RoboDK station: ALTERNATIVA 2 - PYTHON.rdk

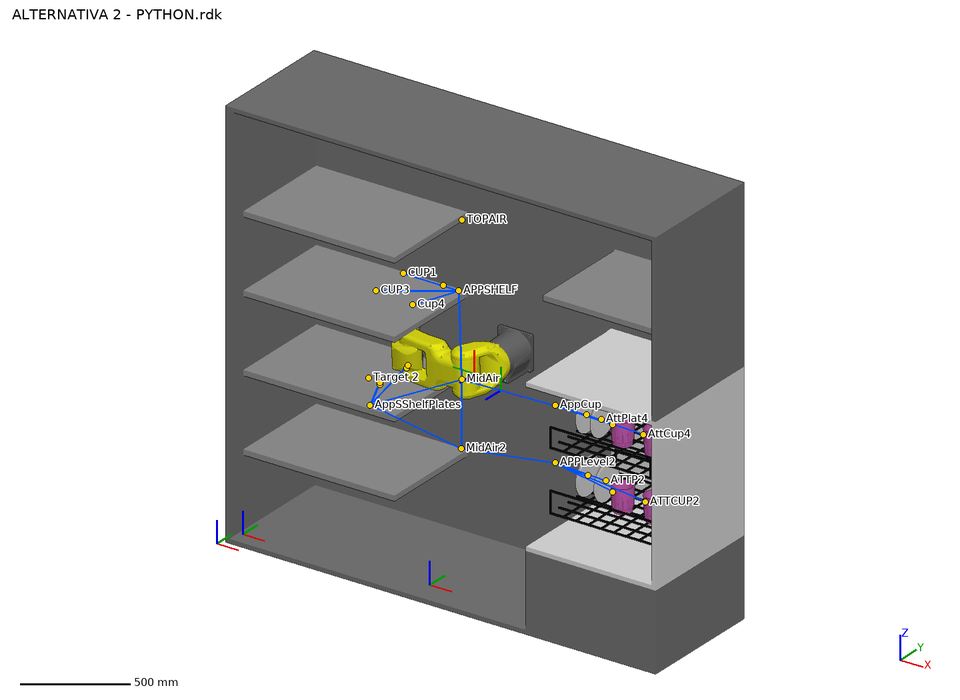
[picture v0: the station drawn from its stored meshes, robots at their saved joint values, targets as dots, program paths as lines]
Station ALTERNATIVA 2 (saved by RoboDK 6.0.0). Poses are relative to the parent item; angles as X-Y-Z fixed-axis rotations.
  - object modelo_solo_interior_v6 at (0, 0, 0) mm, size 2380 x 700 x 2200 mm, geometry from modelo_solo_interior_v6.obj
  - frame MUEBLE  at (-14.91, -46.19, 5.82) mm
  - frame Fanuc LR Mate 200iD Base at (1300, 320, 1000) mm, rotated rx 90 ry 0 rz 0 deg
    - object VASO_2 at (880, -75, 20) mm, size 110.6 x 132.4 x 110.6 mm, geometry from glass-obj.obj
  - frame Frame 3 at (80, 23.81, 50) mm
    - frame My Mechanism Base at (1040, -6.19, 40) mm
      - robot My Mechanism: 1 axes
          modified DH rows (alpha deg, a mm, theta deg, d mm): 0, 0, 0, 0 linear
          base shift (0, 0, 0) mm, rotated rx 180 ry 0 rz 180 deg
          joint limits [0] to [1500]; home [0]; saved at [905.84]
        - frame Fanuc LR Mate 200iD Base at (-120, 180, 120) mm, rotated rx -90 ry 0 rz -180 deg
          - robot Fanuc LR Mate 200iD: 6 axes, payload 7 kg, reach 717 mm, repeatability 0.02 mm, weight 25 kg
              modified DH rows (alpha deg, a mm, theta deg, d mm): 0, 0, 0, 330; -90, 50, -90, 0; 0, 330, 0, 0; -90, 35, 0, 335; 90, 0, 0, 0; -90, 0, 0, 80
              base shift (0, 0, -330) mm
              joint limits [-170, -100, -67, -190, -125, -360] to [170, 145, 213, 190, 124, 360]; home [0, 0, 0, 0, 0, 0]; saved at [93.044, 96.293, -58.546, 87.403, 88.412, -211.418]
            - tool RobotiQ EPick Vacuum Gripper (1 Cup), TCP at (0, 0, 130) mm, size 75 x 83 x 136.1 mm
    - target AttCup4 (Cartesian target) at (2025.95, 272.71, 963.12) mm, rotated rx 90.33 ry 1.97 rz 94.86 deg; joints [-104.637, 115.612, 4.554, 123.155, 17.105, 58.882, 975.84] of Fanuc LR Mate 200iD
    - target AppCup (Cartesian target) at (1576.89, 214.64, 1005.7) mm, rotated rx 96.54 ry 1.97 rz 94.86 deg; joints [-118.032, 21.715, -84.906, 21.706, 80.662, 180.626, 980.84] of Fanuc LR Mate 200iD
    - target Target 2 (Cartesian target) at (718.15, -32.51, 1004.9) mm, rotated rx -83.96 ry 1.97 rz 94.86 deg; joints [109.561, -20.769, -26.684, -42.184, 39.93, -145.464, 905.84] of Fanuc LR Mate 200iD
    - target MidAir (Cartesian target) at (1233.73, -32.54, 1140.54) mm, rotated rx 23.3 ry -5.22 rz 90.43 deg; joints [2.19, -20.76, -26.68, -42.18, 39.92, -145.46, 540.58] of Fanuc LR Mate 200iD
    - target ATTCup3 (Cartesian target) at (1855.95, 272.71, 963.12) mm, rotated rx 90.33 ry 1.97 rz 94.86 deg; joints [-109.413, 54.482, -60.076, 22.825, 57.115, 170.802, 975.84] of Fanuc LR Mate 200iD
    - target AttPlat4 (Cartesian target) at (1791.95, 272.71, 973.12) mm, rotated rx 90.33 ry 1.97 rz 94.86 deg; joints [-110.912, 48.655, -68.61, 22.691, 65.237, 173.884, 975.84] of Fanuc LR Mate 200iD
    - target AttP3 (Cartesian target) at (1710.95, 272.71, 973.12) mm, rotated rx 90.33 ry 1.97 rz 94.86 deg; joints [-115.299, 43.34, -78.431, 25.854, 74.698, 176.966, 975.84] of Fanuc LR Mate 200iD
    - target ATTCUP2 (Cartesian target) at (2035.98, 272.65, 625.36) mm, rotated rx 90.33 ry 1.97 rz 94.86 deg; joints [-104.42, 81.896, -28.227, 32.378, 26.939, 153.732, 637.99] of Fanuc LR Mate 200iD
    - target ATTCUP1 (Cartesian target) at (1855.94, 272.75, 625.32) mm, rotated rx 90.32 ry 1.97 rz 94.87 deg; joints [-109.41, 54.48, -60.08, 22.831, 57.11, 170.799, 637.99] of Fanuc LR Mate 200iD
    - target ATTP2 (Cartesian target) at (1811.98, 282.72, 665.28) mm, rotated rx 90.33 ry 1.97 rz 94.85 deg; joints [-106.543, 51.004, -68.493, 17.943, 64.576, 175.489, 637.99] of Fanuc LR Mate 200iD
    - target ATTP1 (Cartesian target) at (1711.98, 282.72, 665.28) mm, rotated rx 90.33 ry 1.97 rz 94.85 deg; joints [-110.992, 44.665, -81.327, 21.149, 77.053, 178.867, 637.99] of Fanuc LR Mate 200iD
    - target APPLevel2 (Cartesian target) at (1576.9, 214.61, 716.41) mm, rotated rx 96.54 ry 1.97 rz 94.85 deg; joints [-118.03, 21.71, -84.9, 21.7, 80.66, 180.62, 691.56] of Fanuc LR Mate 200iD
    - target CUP1 (Cartesian target) at (548.14, 487.49, 1274.9) mm, rotated rx 90 ry 0 rz -90 deg; joints [120.418, 87.929, -81.134, -30.72, 82.362, 4.516, 1350.84] of Fanuc LR Mate 200iD
    - target MidAir2 (Cartesian target) at (1233.71, -32.66, 789.98) mm, rotated rx 23.3 ry -5.22 rz 90.42 deg; joints [2.19, -20.75, -26.67, -42.17, 39.92, -145.45, 189.94] of Fanuc LR Mate 200iD
    - target APPSHELF (Cartesian target) at (938.14, 367.49, 1344.9) mm, rotated rx 90 ry 0 rz -90 deg; joints [-4.087, -66.431, 278.847, -85.961, -90.628, 171.175, 1350.84] of Fanuc LR Mate 200iD
    - target CUP2 (Cartesian target) at (768.14, 487.49, 1274.9) mm, rotated rx 90 ry 0 rz -90 deg; joints [-37.624, -86.068, 260.858, -52.729, -84.434, 187.263, 1350.84] of Fanuc LR Mate 200iD
    - target Cup4 (Cartesian target) at (768.14, 247.49, 1274.9) mm, rotated rx 90 ry 0 rz -90 deg; joints [142.376, 37.971, -88.312, -52.388, 88.969, 1.337, 1350.84] of Fanuc LR Mate 200iD
    - target CUP3 (Cartesian target) at (548.14, 267.49, 1274.9) mm, rotated rx 90 ry 0 rz -90 deg; joints [120.418, 51.735, -68.201, -32.307, 71.323, 11.448, 1350.84] of Fanuc LR Mate 200iD
    - target TOPAIR (Cartesian target) at (1233.79, -32.51, 1944.12) mm, rotated rx 23.31 ry -5.21 rz 90.43 deg; joints [2.18, -20.76, -26.68, -42.18, 39.91, -145.45, 1344.16] of Fanuc LR Mate 200iD
    - target Plat1 (Cartesian target) at (578.15, 467.49, 814.9) mm, rotated rx 180 ry 0 rz 90 deg; joints [94.025, 94.502, -58.622, 86.562, 87.906, -211.315, 905.84] of Fanuc LR Mate 200iD
    - target Plat2 (Cartesian target) at (578.15, 477.49, 824.9) mm, rotated rx 180 ry 0 rz 90 deg; joints [93.044, 96.293, -58.546, 87.403, 88.412, -211.418, 905.84] of Fanuc LR Mate 200iD
    - target plat3 (Cartesian target) at (578.15, 257.49, 814.9) mm, rotated rx 180 ry 0 rz 90 deg; joints [94.025, 62.542, -50.409, 86.896, 87.436, -219.521, 905.84] of Fanuc LR Mate 200iD
    - target Plat4 (Cartesian target) at (578.15, 257.49, 824.9) mm, rotated rx 180 ry 0 rz 90 deg; joints [93.044, 62.461, -50.507, 87.65, 88.065, -219.453, 905.84] of Fanuc LR Mate 200iD
    - target AppSShelfPlates (Cartesian target) at (773.4, -98.39, 907.8) mm, rotated rx -179.99 ry 0 rz 90.01 deg; joints [82.343, 1.423, -15.826, 92.1, 97.355, -254.032, 905.83] of Fanuc LR Mate 200iD
  - program Attach (3 instructions, listed below)
  - program Detach (3 instructions, listed below)
  - program RecallPosition (1 instructions, listed below)
  - program Prog4 (87 instructions, listed below)
  - Python program Prog5 (listed below)
  - object PLATO1 at (1800, 300, 1040) mm, rotated rx -90 ry 0 rz 90 deg, size 200 x 200 x 4 mm, geometry from tinker.obj
  - object PLATO2 at (1880, 300, 1040) mm, rotated rx -90 ry 0 rz 90 deg, size 200 x 200 x 4 mm, geometry from tinker.obj
  - object PLATO3 at (1900.09, 300, 721.16) mm, rotated rx -90 ry 0 rz 90 deg, size 200 x 200 x 4 mm, geometry from tinker.obj
  - object PLATO4 at (1800, 300, 721.16) mm, rotated rx -90 ry 0 rz 90 deg, size 200 x 200 x 4 mm, geometry from tinker.obj
  - object VASO_1 at (2000, 300, 925) mm, rotated rx 90 ry 0 rz 0 deg, size 110.6 x 132.4 x 110.6 mm, geometry from glass-obj.obj
  - object VASO_3 at (2000, 300, 590) mm, rotated rx 90 ry 0 rz 0 deg, size 110.6 x 132.4 x 110.6 mm, geometry from glass-obj.obj
  - object VASO_4 at (2180, 300, 590) mm, rotated rx 90 ry 0 rz 0 deg, size 110.6 x 132.4 x 110.6 mm, geometry from glass-obj.obj
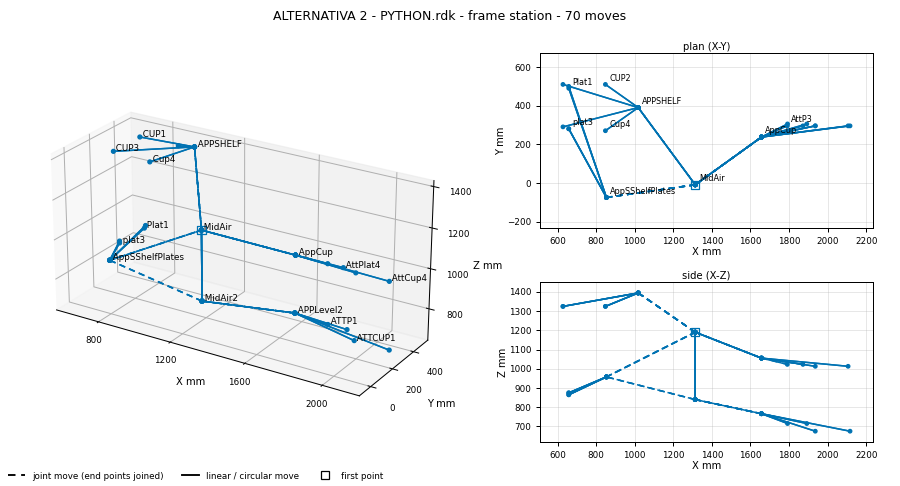
[picture p0: tool path of ALTERNATIVA 2 - PYTHON.rdk in frame station, 70 of 70 moves have a stored position in this frame; points joined in program order, loops and branches not executed]

--- program Attach (robot Fanuc LR Mate 200iD) ---
  Set Ref.: Frame 3
  Set Tool: RobotiQ EPick Vacuum Gripper (1 Cup)
  Attach to RobotiQ EPick Vacuum Gripper (1 Cup)

--- program Detach (robot Fanuc LR Mate 200iD) ---
  Set Ref.: Frame 3
  Set Tool: RobotiQ EPick Vacuum Gripper (1 Cup)
  Detach from RobotiQ EPick Vacuum Gripper (1 Cup)

--- program RecallPosition ---
  Move objects

--- program Prog4 (robot Fanuc LR Mate 200iD) ---
  Set Ref.: Frame 3
  MoveJ (MidAir)
  MoveJ (AppCup)
  MoveJ (AttP3)
  Call Attach
  MoveL (AppCup)
  MoveL (MidAir)
  MoveJ (AppSShelfPlates)
  MoveL (Plat1)
  Call Detach
  MoveL (AppSShelfPlates)
  MoveJ (MidAir)
  MoveJ (AppCup)
  MoveL (AttPlat4)
  Call Attach
  MoveL (AppCup)
  MoveL (MidAir)
  MoveJ (AppSShelfPlates)
  MoveL (Plat2)
  Call Detach
  MoveL (AppSShelfPlates)
  MoveJ (MidAir)
  MoveL (MidAir2)
  MoveJ (APPLevel2)
  MoveL (ATTP1)
  Call Attach
  MoveL (APPLevel2)
  MoveJ (MidAir2)
  MoveJ (AppSShelfPlates)
  MoveL (plat3)
  Call Detach
  MoveL (AppSShelfPlates)
  MoveJ (MidAir2)
  MoveJ (APPLevel2)
  MoveL (ATTP2)
  Call Attach
  MoveL (APPLevel2)
  MoveJ (MidAir2)
  MoveJ (AppSShelfPlates)
  MoveL (Plat4)
  Call Detach
  MoveL (AppSShelfPlates)
  MoveJ (MidAir)
  MoveJ (AppCup)
  MoveL (ATTCup3)
  Call Attach
  MoveL (AppCup)
  MoveL (MidAir)
  MoveJ (APPSHELF)
  MoveL (CUP1)
  Call Detach
  MoveL (APPSHELF)
  MoveJ (MidAir)
  MoveJ (AppCup)
  MoveL (AttCup4)
  Call Attach
  MoveL (AppCup)
  MoveL (MidAir)
  MoveJ (APPSHELF)
  MoveL (CUP2)
  Call Detach
  MoveL (APPSHELF)
  MoveJ (MidAir)
  MoveL (MidAir2)
  MoveJ (APPLevel2)
  MoveL (ATTCUP1)
  Call Attach
  MoveL (APPLevel2)
  MoveJ (MidAir2)
  MoveL (MidAir)
  MoveJ (APPSHELF)
  MoveL (CUP3)
  Call Detach
  MoveL (APPSHELF)
  MoveJ (MidAir)
  MoveL (MidAir2)
  MoveJ (APPLevel2)
  MoveL (ATTCUP2)
  Call Attach
  MoveL (APPLevel2)
  MoveL (MidAir2)
  MoveL (MidAir)
  MoveJ (APPSHELF)
  MoveL (Cup4)
  Call Detach
  MoveL (APPSHELF)
  MoveJ (MidAir)

--- Python program Prog5 ---
# ============================================================
# ANALISIS ROBODK - Prog4
#
# Datos mostrados:
# - Programa analizado
# - Tiempo ciclo
# - Distancia recorrida por el TCP en mm y m
# - Instrucciones válidas
# - Total de instrucciones
# - Total de movimientos
# - Nº MoveJ
# - Nº MoveL
# ============================================================

import os
import csv
import datetime

try:
    from robodk.robolink import *
except:
    from robolink import *


# ================= CONFIGURACIÓN =================

PROGRAMA = "Prog4"
EXPORTAR_CSV = True


# ================= CONEXIÓN CON ROBODK =================

RDK = Robolink()

prog = RDK.Item(PROGRAMA, ITEM_TYPE_PROGRAM)

if not prog.Valid():
    RDK.ShowMessage("No se ha encontrado el programa: " + PROGRAMA)
    raise Exception("No se ha encontrado el programa: " + PROGRAMA)


# ================= DATOS DE TIEMPO Y DISTANCIA =================

try:
    resultado_update = prog.Update(COLLISION_ON, 3600)

    instrucciones_validas = int(resultado_update[0])
    tiempo_ciclo_s = float(resultado_update[1])
    distancia_tcp_mm = float(resultado_update[2])

except Exception as e:
    instrucciones_validas = 0
    tiempo_ciclo_s = 0.0
    distancia_tcp_mm = 0.0
    RDK.ShowMessage("Error al actualizar el programa: " + str(e))


distancia_tcp_m = distancia_tcp_mm / 1000.0


# ================= CONTAR MOVIMIENTOS =================

total_instrucciones = prog.InstructionCount()

total_movimientos = 0
num_movej = 0
num_movel = 0

for i in range(total_instrucciones):

    try:
        nombre, instype, movetype, es_target_articular, pose, joints = prog.Instruction(i)
    except:
        continue

    if instype == INS_TYPE_MOVE:

        total_movimientos += 1

        if movetype == MOVE_TYPE_JOINT:
            num_movej += 1

        elif movetype == MOVE_TYPE_LINEAR:
            num_movel += 1


# ================= MOSTRAR RESULTADOS =================

mensaje = ""
mensaje += "RESULTADOS DEL PROGRAMA ROBODK\n"
mensaje += "====================================\n\n"

mensaje += "Programa analizado: {}\n".format(prog.Name())
mensaje += "Tiempo ciclo: {:.3f} s\n".format(tiempo_ciclo_s)
mensaje += "Distancia recorrida por el TCP: {:.3f} mm\n".format(distancia_tcp_mm)
mensaje += "Distancia recorrida por el TCP: {:.3f} m\n".format(distancia_tcp_m)
mensaje += "Instrucciones válidas: {}\n".format(instrucciones_validas)
mensaje += "Total de instrucciones: {}\n".format(total_instrucciones)
mensaje += "Total de movimientos: {}\n".format(total_movimientos)
mensaje += "Nº MoveJ: {}\n".format(num_movej)
mensaje += "Nº MoveL: {}\n".format(num_movel)

print(mensaje)
RDK.ShowMessage(mensaje)


# ================= EXPORTAR A CSV =================

if EXPORTAR_CSV:

    escritorio = os.path.join(os.path.expanduser("~"), "Desktop")
    ruta_csv = os.path.join(escritorio, "resultados_robodk_Prog4.csv")

    if not os.path.isdir(escritorio):
        ruta_csv = os.path.join(os.getcwd(), "resultados_robodk_Prog4.csv")

    existe_archivo = os.path.isfile(ruta_csv)

    with open(ruta_csv, mode="a", newline="", encoding="utf-8-sig") as archivo:
        writer = csv.writer(archivo, delimiter=";")

        if not existe_archivo:
            writer.writerow([
                "Fecha",
                "Programa analizado",
                "Tiempo ciclo (s)",
                "Distancia TCP (mm)",
                "Distancia TCP (m)",
                "Instrucciones validas",
                "Total instrucciones",
                "Total movimientos",
                "MoveJ",
                "MoveL"
            ])

        writer.writerow([
            datetime.datetime.now().strftime("%Y-%m-%d %H:%M:%S"),
            prog.Name(),
            round(tiempo_ciclo_s, 3),
            round(distancia_tcp_mm, 3),
            round(distancia_tcp_m, 3),
            instrucciones_validas,
            total_instrucciones,
            total_movimientos,
            num_movej,
            num_movel
        ])

    print("\nCSV guardado en:")
    print(ruta_csv)
